{attribute 'linkalways'} 
{attribute 'no_explicit_call' := 'This FB is a CLASS and must be accessed using methods or properties'}
{attribute 'enable_dynamic_creation'}
FUNCTION_BLOCK JsonDeserializerChangedEvent EXTENDS JsonDeserializerEvent IMPLEMENTS I_JsonDeserializerChangedEvent

END_FUNCTION_BLOCK

(* stored: Version 1.1.0.1, ProductVersion 3.1.4024.12
   POU JsonDeserializerChangedEvent: Id {67468afd-548e-4069-9d80-12a3de2c4b14}, SpecialFunc None *)
